// TIA Portal V18 export
// export: Created 2026-01-09T11:32:00.750215Z, ExportSetting WithDefaults, DisplayName Totally Integrated Automation Portal, DisplayVersion V18 Update 5, DisplayName TIA Portal Openness, DisplayVersion V18 Update 5, DisplayName TIA Portal Teamcenter Gateway, DisplayVersion V18, DisplayName TIA Portal Version Control Interface, DisplayVersion V18, DisplayName SINAMICS Startdrive Advanced, DisplayVersion V18 SP2 Update 1, DisplayName SINAMICS Startdrive G110M, G120, G120C, G120D, G120P, G115D, DisplayVersion V18 SP2 Update 1, DisplayName SINAMICS Startdrive G130, G150, S120, S150, SINAMICS MV, S210, G220, S200, DisplayVersion V18 SP2 Update 1, DisplayName STEP 7 Professional, DisplayVersion V18 Update 5, DisplayName STEP 7 Safety, DisplayVersion V18, DisplayName WinCC Professional, DisplayVersion V18 Update 5
TagTable "SR_X80"
  KeyenceSR1000Ctrl_800A1DB_sHMI : RCS_KeyenceSR1000_HMI1  (PLC tag KeyenceSR1000Ctrl_800A1DB.sHMI, CPU S71500-2PN_TP700, 1 s)
    TagStructureMember "Manual"
      TagStructureMember "Preset"
      TagStructureMember "Trigger"
    TagStructureMember "Status"
      TagStructureMember "Ready"
      TagStructureMember "Busy"
      TagStructureMember "Failure"
      TagStructureMember "Complete"
      TagStructureMember "ReadOk"
      TagStructureMember "ReadNok"
      TagStructureMember "TimeOut"
      TagStructureMember "Error"
      TagStructureMember "ErrorCode"
      TagStructureMember "Sequence"
      TagStructureMember "iReTriggerTimes"
      TagStructureMember "CurrentLength"
      TagStructureMember "CurrentCode"
      TagStructureMember "LastCode"
    TagStructureMember "Indata"
      TagStructureMember "ReadComplete"
      TagStructureMember "ReadFailure"
      TagStructureMember "GeneralErrorCode"
      TagStructureMember "ReadResultCode"
      TagStructureMember "ResultDataSize"
    TagStructureMember "Outdata"
      TagStructureMember "ReadCompleteClear"
      TagStructureMember "ErrorClear"
      TagStructureMember "ReadRequest"
  KeyenceSR1000Ctrl_801A1DB_sHMI : RCS_KeyenceSR1000_HMI1  (PLC tag KeyenceSR1000Ctrl_801A1DB.sHMI, CPU S71500-2PN_TP700, 1 s)
    TagStructureMember "Manual"
      TagStructureMember "Preset"
      TagStructureMember "Trigger"
    TagStructureMember "Status"
      TagStructureMember "Ready"
      TagStructureMember "Busy"
      TagStructureMember "Failure"
      TagStructureMember "Complete"
      TagStructureMember "ReadOk"
      TagStructureMember "ReadNok"
      TagStructureMember "TimeOut"
      TagStructureMember "Error"
      TagStructureMember "ErrorCode"
      TagStructureMember "Sequence"
      TagStructureMember "iReTriggerTimes"
      TagStructureMember "CurrentLength"
      TagStructureMember "CurrentCode"
      TagStructureMember "LastCode"
    TagStructureMember "Indata"
      TagStructureMember "ReadComplete"
      TagStructureMember "ReadFailure"
      TagStructureMember "GeneralErrorCode"
      TagStructureMember "ReadResultCode"
      TagStructureMember "ResultDataSize"
    TagStructureMember "Outdata"
      TagStructureMember "ReadCompleteClear"
      TagStructureMember "ErrorClear"
      TagStructureMember "ReadRequest"
  KeyenceSR1000Ctrl_802A1DB_sHMI : RCS_KeyenceSR1000_HMI1  (PLC tag KeyenceSR1000Ctrl_802A1DB.sHMI, CPU S71500-2PN_TP700, 1 s)
    TagStructureMember "Manual"
      TagStructureMember "Preset"
      TagStructureMember "Trigger"
    TagStructureMember "Status"
      TagStructureMember "Ready"
      TagStructureMember "Busy"
      TagStructureMember "Failure"
      TagStructureMember "Complete"
      TagStructureMember "ReadOk"
      TagStructureMember "ReadNok"
      TagStructureMember "TimeOut"
      TagStructureMember "Error"
      TagStructureMember "ErrorCode"
      TagStructureMember "Sequence"
      TagStructureMember "iReTriggerTimes"
      TagStructureMember "CurrentLength"
      TagStructureMember "CurrentCode"
      TagStructureMember "LastCode"
    TagStructureMember "Indata"
      TagStructureMember "ReadComplete"
      TagStructureMember "ReadFailure"
      TagStructureMember "GeneralErrorCode"
      TagStructureMember "ReadResultCode"
      TagStructureMember "ResultDataSize"
    TagStructureMember "Outdata"
      TagStructureMember "ReadCompleteClear"
      TagStructureMember "ErrorClear"
      TagStructureMember "ReadRequest"
  KeyenceSR1000Ctrl_803A1DB_sHMI : RCS_KeyenceSR1000_HMI1  (PLC tag KeyenceSR1000Ctrl_803A1DB.sHMI, CPU S71500-2PN_TP700, 1 s)
    TagStructureMember "Manual"
      TagStructureMember "Preset"
      TagStructureMember "Trigger"
    TagStructureMember "Status"
      TagStructureMember "Ready"
      TagStructureMember "Busy"
      TagStructureMember "Failure"
      TagStructureMember "Complete"
      TagStructureMember "ReadOk"
      TagStructureMember "ReadNok"
      TagStructureMember "TimeOut"
      TagStructureMember "Error"
      TagStructureMember "ErrorCode"
      TagStructureMember "Sequence"
      TagStructureMember "iReTriggerTimes"
      TagStructureMember "CurrentLength"
      TagStructureMember "CurrentCode"
      TagStructureMember "LastCode"
    TagStructureMember "Indata"
      TagStructureMember "ReadComplete"
      TagStructureMember "ReadFailure"
      TagStructureMember "GeneralErrorCode"
      TagStructureMember "ReadResultCode"
      TagStructureMember "ResultDataSize"
    TagStructureMember "Outdata"
      TagStructureMember "ReadCompleteClear"
      TagStructureMember "ErrorClear"
      TagStructureMember "ReadRequest"
  KeyenceSR1000Ctrl_804A1DB_sHMI : RCS_KeyenceSR1000_HMI1  (PLC tag KeyenceSR1000Ctrl_804A1DB.sHMI, CPU S71500-2PN_TP700, 1 s)
    TagStructureMember "Manual"
      TagStructureMember "Preset"
      TagStructureMember "Trigger"
    TagStructureMember "Status"
      TagStructureMember "Ready"
      TagStructureMember "Busy"
      TagStructureMember "Failure"
      TagStructureMember "Complete"
      TagStructureMember "ReadOk"
      TagStructureMember "ReadNok"
      TagStructureMember "TimeOut"
      TagStructureMember "Error"
      TagStructureMember "ErrorCode"
      TagStructureMember "Sequence"
      TagStructureMember "iReTriggerTimes"
      TagStructureMember "CurrentLength"
      TagStructureMember "CurrentCode"
      TagStructureMember "LastCode"
    TagStructureMember "Indata"
      TagStructureMember "ReadComplete"
      TagStructureMember "ReadFailure"
      TagStructureMember "GeneralErrorCode"
      TagStructureMember "ReadResultCode"
      TagStructureMember "ResultDataSize"
    TagStructureMember "Outdata"
      TagStructureMember "ReadCompleteClear"
      TagStructureMember "ErrorClear"
      TagStructureMember "ReadRequest"
  KeyenceSR1000Ctrl_805A1DB_sHMI : RCS_KeyenceSR1000_HMI1  (PLC tag KeyenceSR1000Ctrl_805A1DB.sHMI, CPU S71500-2PN_TP700, 1 s)
    TagStructureMember "Manual"
      TagStructureMember "Preset"
      TagStructureMember "Trigger"
    TagStructureMember "Status"
      TagStructureMember "Ready"
      TagStructureMember "Busy"
      TagStructureMember "Failure"
      TagStructureMember "Complete"
      TagStructureMember "ReadOk"
      TagStructureMember "ReadNok"
      TagStructureMember "TimeOut"
      TagStructureMember "Error"
      TagStructureMember "ErrorCode"
      TagStructureMember "Sequence"
      TagStructureMember "iReTriggerTimes"
      TagStructureMember "CurrentLength"
      TagStructureMember "CurrentCode"
      TagStructureMember "LastCode"
    TagStructureMember "Indata"
      TagStructureMember "ReadComplete"
      TagStructureMember "ReadFailure"
      TagStructureMember "GeneralErrorCode"
      TagStructureMember "ReadResultCode"
      TagStructureMember "ResultDataSize"
    TagStructureMember "Outdata"
      TagStructureMember "ReadCompleteClear"
      TagStructureMember "ErrorClear"
      TagStructureMember "ReadRequest"
  KeyenceSR1000Ctrl_806A1DB_sHMI : RCS_KeyenceSR1000_HMI1  (PLC tag KeyenceSR1000Ctrl_806A1DB.sHMI, CPU S71500-2PN_TP700, 1 s)
    TagStructureMember "Manual"
      TagStructureMember "Preset"
      TagStructureMember "Trigger"
    TagStructureMember "Status"
      TagStructureMember "Ready"
      TagStructureMember "Busy"
      TagStructureMember "Failure"
      TagStructureMember "Complete"
      TagStructureMember "ReadOk"
      TagStructureMember "ReadNok"
      TagStructureMember "TimeOut"
      TagStructureMember "Error"
      TagStructureMember "ErrorCode"
      TagStructureMember "Sequence"
      TagStructureMember "iReTriggerTimes"
      TagStructureMember "CurrentLength"
      TagStructureMember "CurrentCode"
      TagStructureMember "LastCode"
    TagStructureMember "Indata"
      TagStructureMember "ReadComplete"
      TagStructureMember "ReadFailure"
      TagStructureMember "GeneralErrorCode"
      TagStructureMember "ReadResultCode"
      TagStructureMember "ResultDataSize"
    TagStructureMember "Outdata"
      TagStructureMember "ReadCompleteClear"
      TagStructureMember "ErrorClear"
      TagStructureMember "ReadRequest"
  KeyenceSR1000Ctrl_807A1DB_sHMI : RCS_KeyenceSR1000_HMI1  (PLC tag KeyenceSR1000Ctrl_807A1DB.sHMI, CPU S71500-2PN_TP700, 1 s)
    TagStructureMember "Manual"
      TagStructureMember "Preset"
      TagStructureMember "Trigger"
    TagStructureMember "Status"
      TagStructureMember "Ready"
      TagStructureMember "Busy"
      TagStructureMember "Failure"
      TagStructureMember "Complete"
      TagStructureMember "ReadOk"
      TagStructureMember "ReadNok"
      TagStructureMember "TimeOut"
      TagStructureMember "Error"
      TagStructureMember "ErrorCode"
      TagStructureMember "Sequence"
      TagStructureMember "iReTriggerTimes"
      TagStructureMember "CurrentLength"
      TagStructureMember "CurrentCode"
      TagStructureMember "LastCode"
    TagStructureMember "Indata"
      TagStructureMember "ReadComplete"
      TagStructureMember "ReadFailure"
      TagStructureMember "GeneralErrorCode"
      TagStructureMember "ReadResultCode"
      TagStructureMember "ResultDataSize"
    TagStructureMember "Outdata"
      TagStructureMember "ReadCompleteClear"
      TagStructureMember "ErrorClear"
      TagStructureMember "ReadRequest"
